KUKA KRL data list: kuka_eki_command_serverB.dat

&ACCESS RVO1
&PARAM EDITMASK = *
&PARAM TEMPLATE = C:\KRC\Roboter\Template\submit
defdat kuka_eki_command_serverB public
;FOLD EXTERNAL DECLARATIONS;%{PE}%MKUKATPBASIS,%CEXT,%VCOMMON,%P
;FOLD BASISTECH EXT;%{PE}%MKUKATPBASIS,%CEXT,%VEXT,%P
EXT  BAS (BAS_COMMAND  :IN,REAL  :IN )
DECL INT SUCCESS
;ENDFOLD (BASISTECH EXT)
;FOLD USER EXT;%{E}%MKUKATPUSER,%CEXT,%VEXT,%P
;Make your modifications here

;ENDFOLD (USER EXT)
;ENDFOLD (EXTERNAL DECLARATIONS)
decl global INT instruction_code = 0          ; identify which command (i.e, velocity, motion, laser, etc)
decl global real parameters[6]                ; number of received parameters in real value
decl global real json_motion_complete = 0     ; json motion command complete or not
decl global real wait_time = 0                ; wait time between move
parameters[1] = 0
decl global frame cartesian_target            ; frame is a sturct, X, Y, Z, A, B, C
;decl global pos cartesian_target_pos          ;pos: X, Y, Z, A, B, C, INT S, T
enddat
